Fanuc TP program (LS listing): edited_fixA.ls

/PROG MOVE_P2
/ATTR
OWNER = MNEDITOR;
COMMENT = "auto";
/MN
   1:  UFRAME_NUM=1 ;
   2:  UTOOL_NUM=1 ;
   3:  !edited: final move now goes to fixture A place ;
   4:  J PR[1:home] 100% FINE ;
   5:  L PR[8:fixture A place] 100mm/sec FINE ;
/POS
/END
